(* CODESYS project Tc3_Physics.library
   TcLibraryId: Beckhoff Automation GmbH|Tc3_Physics|3.4.67.0
   Company: Beckhoff Automation GmbH
   DefaultNamespace: Tc3_Physics
   Version: 3.4.67.0
   Placeholder: Tc3_Physics
   Title: Tc3_Physics

Project tree, tasks and I/O mapping:
  Version/
    global variables Global_Version
  POUs/
    _Internal/
      function block IPlcGeometry2D [ST]: FB_init, FB_exit
      function block IPlcDynamicConstraint [ST]: FB_init, FB_exit
    Spatial/
      Positions/
        function block PositionXY [ST]: FB_init, FB_reinit, FB_exit, SetZero, SetValues, SetValuesXY, SetValuesRP, SetValuesXYReferenceId, GetRadius, GetPhi, Invert, ConcatenateWith, ShiftByXY, x, y, ReferenceId
        function block PositionXYC [ST]: FB_init, FB_reinit, FB_exit, SetZero, SetValues, SetValuesXY, SetValuesXYC, SetValuesXYCReferenceId, Invert, ConcatenateWith, StepByLocalXY, ShiftByXY, TurnByC, Transform, x, y, c, ReferenceId
    Dynamics/
      function block DynamicConstraint_Container [ST]: FB_init, FB_exit, Clear, AddConstraint, AddConstraintByReference, Count
      function block DynamicConstraint_CartesianXY [ST]: FB_init, FB_exit, SetValuesVAJ, V, A, J
      function block DynamicConstraint_CartesianXYZ [ST]: FB_init, FB_exit, SetValuesVAJ, V, A, J
      function block DynamicConstraint_PathXY [ST]: FB_init, FB_exit, SetValuesVADJ, V, A, D, J
      function block DynamicConstraint_PathXYZ [ST]: FB_init, FB_exit, SetValuesVADJ, V, A, D, J
      function block DynamicConstraint_Coordinates [ST]: FB_init, FB_exit, AddLimit, SetLimit, RemoveLimit, Clear, GetV, GetA, GetD, GetJ, Count
    Coordinates/
      function GetMcsCoordinateType [ST]
      function GetUninterpretedCoordinateType [ST]
      function GetAcsCoordinateType [ST]
  DUTs/
    Enumerations/
      data type E_RotationCoordinates
      data type E_CoordCategory
      data type E_McsCoordType
    data type CoordinateType
  GVLs/
    global variables GVL
*)

// DUTs/CoordinateType

(* Coordinate type. Use provided constants such as Coord_Mcs_X or factory functions such as GetMcsCoordinateType for creation. *)
	{attribute 'TcIecLibraryType'}
TYPE CoordinateType : 
	STRUCT
		(* Reserved. *)
		{attribute 'hide'}
		_reserved0 : ULINT := 0;
	END_STRUCT
END_TYPE

// DUTs/Enumerations/E_RotationCoordinates

(* 
    Enumeration of rotation conventions. 
    The order of letters defines the order of rotation around local axes.
    This also defines order in which user should program rotation values.
   *)
	{attribute 'TcIecLibraryType'}
{attribute 'qualified_only'}
{attribute 'strict'}
{attribute 'to_string'}
TYPE E_RotationCoordinates : (
	ABC:=0, 	(* ABC *)
	ACB:=1, 	(* ACB *)
	BCA:=2, 	(* BCA *)
	BAC:=3, 	(* BAC *)
	CAB:=4, 	(* CAB *)
	CBA:=5, 	(* CBA *)
	ABA:=6, 	(* ABA *)
	ACA:=7, 	(* ACA *)
	BCB:=8, 	(* BCB *)
	BAB:=9, 	(* BAB *)
	CAC:=10, 	(* CAC *)
	CBC:=11	(* CBC *)
) UDINT;
END_TYPE

// DUTs/Enumerations/E_CoordCategory

(* 
    Enumeration coordinate categories.
   *)
	{attribute 'TcIecLibraryType'}
{attribute 'qualified_only'}
{attribute 'strict'}
{attribute 'to_string'}
TYPE E_CoordCategory : (
	Invalid:=16#0, 	(* Invalid *)
	MCS:=16#1, 	(* MCS *)
	ACS:=16#2, 	(* ACS *)
	Uninterpreted:=16#3	(* Uninterpreted *)
) UDINT;
END_TYPE

// DUTs/Enumerations/E_McsCoordType

(* 
    Enumeration of MCS coordinate types.
   *)
	{attribute 'TcIecLibraryType'}
{attribute 'qualified_only'}
{attribute 'strict'}
{attribute 'to_string'}
TYPE E_McsCoordType : (
	Invalid:=16#0, 	(* Invalid *)
	X:=16#11, 	(* X *)
	Y:=16#21, 	(* Y *)
	Z:=16#31, 	(* Z *)
	A1:=16#41, 	(* A1 *)
	A2:=16#42, 	(* A2 *)
	A3:=16#43, 	(* A3 *)
	B1:=16#51, 	(* B1 *)
	B2:=16#52, 	(* B2 *)
	B3:=16#53, 	(* B3 *)
	C1:=16#61, 	(* C1 *)
	C2:=16#62, 	(* C2 *)
	C3:=16#63	(* C3 *)
) UDINT;
END_TYPE

// Version/Global_Version
{attribute 'TcGenerated'}
// This function has been automatically generated from the project information.
VAR_GLOBAL CONSTANT
	{attribute 'const_non_replaced'}
	{attribute 'linkalways'}
	stLibVersion_Tc3_Physics : ST_LibVersion := (iMajor := 3, iMinor := 4, iBuild := 67, iRevision := 0, sVersion := '3.4.67.0');
	{attribute 'const_non_replaced'}
	{attribute 'linkalways'}
	sLibraryId_Tc3_Physics : String := 'Beckhoff Automation GmbH|Tc3_Physics|3.4.67.0';
END_VAR

// GVLs/GVL

	{attribute 'external_name' := 'GVL_GUID_33C55D4C_0C6D_4080_813F_F3548CAD353B'}
VAR_GLOBAL CONSTANT
		Coord_Mcs_X	:	CoordinateType := GetMcsCoordinateType(E_McsCoordType.X);
		Coord_Mcs_Y	:	CoordinateType := GetMcsCoordinateType(E_McsCoordType.Y);
		Coord_Mcs_Z	:	CoordinateType := GetMcsCoordinateType(E_McsCoordType.Z);
		Coord_Mcs_A1	:	CoordinateType := GetMcsCoordinateType(E_McsCoordType.A1);
		Coord_Mcs_A2	:	CoordinateType := GetMcsCoordinateType(E_McsCoordType.A2);
		Coord_Mcs_A3	:	CoordinateType := GetMcsCoordinateType(E_McsCoordType.A3);
		Coord_Mcs_B1	:	CoordinateType := GetMcsCoordinateType(E_McsCoordType.B1);
		Coord_Mcs_B2	:	CoordinateType := GetMcsCoordinateType(E_McsCoordType.B2);
		Coord_Mcs_B3	:	CoordinateType := GetMcsCoordinateType(E_McsCoordType.B3);
		Coord_Mcs_C1	:	CoordinateType := GetMcsCoordinateType(E_McsCoordType.C1);
		Coord_Mcs_C2	:	CoordinateType := GetMcsCoordinateType(E_McsCoordType.C2);
		Coord_Mcs_C3	:	CoordinateType := GetMcsCoordinateType(E_McsCoordType.C3);
		Coord_Uninterpreted1	:	CoordinateType := GetUninterpretedCoordinateType(1);
		Coord_Uninterpreted2	:	CoordinateType := GetUninterpretedCoordinateType(2);
		Coord_Uninterpreted3	:	CoordinateType := GetUninterpretedCoordinateType(3);
		Coord_Uninterpreted4	:	CoordinateType := GetUninterpretedCoordinateType(4);
		Coord_Uninterpreted5	:	CoordinateType := GetUninterpretedCoordinateType(5);
		Coord_Uninterpreted6	:	CoordinateType := GetUninterpretedCoordinateType(6);
		Coord_Uninterpreted7	:	CoordinateType := GetUninterpretedCoordinateType(7);
		Coord_Uninterpreted8	:	CoordinateType := GetUninterpretedCoordinateType(8);
		Coord_Acs1	:	CoordinateType := GetAcsCoordinateType(1);
		Coord_Acs2	:	CoordinateType := GetAcsCoordinateType(2);
		Coord_Acs3	:	CoordinateType := GetAcsCoordinateType(3);
		Coord_Acs4	:	CoordinateType := GetAcsCoordinateType(4);
		Coord_Acs5	:	CoordinateType := GetAcsCoordinateType(5);
		Coord_Acs6	:	CoordinateType := GetAcsCoordinateType(6);
	END_VAR

// POUs/_Internal/IPlcGeometry2D

	{attribute 'c++_compatible'}
	{attribute 'external_name' := 'IPlcGeometry2D_GUID_432B7521_EF05_1C03_897A_3B970F77C0D6'}
	{attribute 'TcIecLibraryType'}
	{attribute 'no_explicit_call' :='do not call this POU directly'}
	{attribute 'no_assign_warning'}
	(* Internal representation of an object in the planar space. *)
	FUNCTION_BLOCK IPlcGeometry2D
	VAR
		(* x-coordinate of the instance. *)
		px : LREAL;
		(* y-coordinate of the instance. *)
		py : LREAL;
		(* c-rotation of the instance given in degrees [°]. *)
		pc : LREAL;
		 {attribute 'hide'}
		_reserved1 : ARRAY [1..24] OF USINT;
	END_VAR
	VAR_OUTPUT
		(* ErrorCode for last method execution *)
		nErrorId : UDINT;
		(* Error during last method execution *)
		bError : BOOL;
	END_VAR
	VAR
		 {attribute 'hide'}
		_reserved2 : ARRAY [1..35] OF USINT;
	END_VAR


	(* Internal method *)
	{attribute 'hide'}
	METHOD FB_init : BOOL
	VAR_INPUT
		(*  if TRUE, the retain variables are initialized (warm start / cold start) *)
		bInitRetains : BOOL;
		(*  if TRUE, the instance afterwards gets moved into the copy code (online change) *)
		bInCopyCode : BOOL;
	END_VAR
END_METHOD


	(* Internal method *)
	{attribute 'hide'}
	METHOD FB_exit : BOOL
	VAR_INPUT
		(*  if TRUE, the exit method is called for exiting an instance that is copied afterwards (online change). *)
		bInCopyCode : BOOL;
	END_VAR
END_METHOD

END_FUNCTION_BLOCK

// POUs/_Internal/IPlcDynamicConstraint

	{attribute 'c++_compatible'}
	{attribute 'external_name' := 'IPlcDynamicConstraint_GUID_6C0A73A2_C983_14C5_9BC7_15048F604248'}
	{attribute 'TcIecLibraryType'}
	{attribute 'no_explicit_call' := 'do not call this POU directly'}
	{attribute 'no_assign_warning'}
	(* Internal representation of dynamic constraints. *)
	FUNCTION_BLOCK IPlcDynamicConstraint
	VAR
		{attribute 'hide'}
		_reserved0 : ULINT;
		 {attribute 'hide'}
		_reserved1 : UINT_0_32;
		 {attribute 'hide'}
		_reserved2 : ARRAY [1..4] OF UINT_8_16;
		 {attribute 'hide'}
		_reserved3 : ARRAY [1..20] OF USINT;
	END_VAR


	(* Internal method *)
	{attribute 'hide'}
	METHOD FB_init : BOOL
	VAR_INPUT
		(*  if TRUE, the retain variables are initialized (warm start / cold start) *)
		bInitRetains : BOOL;
		(*  if TRUE, the instance afterwards gets moved into the copy code (online change) *)
		bInCopyCode : BOOL;
	END_VAR
END_METHOD


	(* Internal method *)
	{attribute 'hide'}
	METHOD FB_exit : BOOL
	VAR_INPUT
		(*  if TRUE, the exit method is called for exiting an instance that is copied afterwards (online change). *)
		bInCopyCode : BOOL;
	END_VAR
END_METHOD

END_FUNCTION_BLOCK

// POUs/Dynamics/DynamicConstraint_Container

	{attribute 'c++_compatible'}
	{attribute 'external_name' := 'DynamicConstraint_Container_GUID_0829228B_5233_1C1E_8F00_79BA3B649C7B'}
	{attribute 'TcIecLibraryType'}
	{attribute 'no_explicit_call' := 'do not call this POU directly'}
	{attribute 'no_assign_warning'}
	(* A container for dynamic constraints. *)
	FUNCTION_BLOCK DynamicConstraint_Container EXTENDS IPlcDynamicConstraint


	(* Internal method *)
	{attribute 'hide'}
	METHOD FB_init : BOOL
	VAR_INPUT
		(*  if TRUE, the retain variables are initialized (warm start / cold start) *)
		bInitRetains : BOOL;
		(*  if TRUE, the instance afterwards gets moved into the copy code (online change) *)
		bInCopyCode : BOOL;
	END_VAR
END_METHOD


	(* Internal method *)
	{attribute 'hide'}
	METHOD FB_exit : BOOL
	VAR_INPUT
		(*  if TRUE, the exit method is called for exiting an instance that is copied afterwards (online change). *)
		bInCopyCode : BOOL;
	END_VAR
END_METHOD


	(* Removes all dynamic constraints from the container. *)
	METHOD Clear
END_METHOD


	(* Adds a copy of a dynamic constraint to the container. If the dynamic constraint changes afterwards, the value in the container will not reflect that change. *)
	METHOD AddConstraint
	VAR_INPUT
		(* A reference to the constraint to be added. *)
 {attribute 'GUID' := '6C0A73A2-C983-14C5-9BC7-15048F604248'}
				Constraint : REFERENCE TO IPlcDynamicConstraint;
	END_VAR
END_METHOD


	(* Adds a reference to a dynamic constraint to the container. If the dynamic constraint changes afterwards, the value in the container will reflect that change. *)
	METHOD AddConstraintByReference
	VAR_INPUT
		(* A reference to the constraint to be added. *)
 {attribute 'GUID' := '6C0A73A2-C983-14C5-9BC7-15048F604248'}
				Constraint : REFERENCE TO IPlcDynamicConstraint;
	END_VAR
END_METHOD


{attribute 'monitoring' := 'call'}
	PROPERTY Count : UDINT
GET
END_GET
END_PROPERTY

END_FUNCTION_BLOCK

// POUs/Dynamics/DynamicConstraint_CartesianXY

	{attribute 'c++_compatible'}
	{attribute 'external_name' := 'DynamicConstraint_CartesianXY_GUID_45D77D0C_DF69_1CCA_AAA6_5FE79B258E7C'}
	{attribute 'TcIecLibraryType'}
	{attribute 'no_explicit_call' := 'do not call this POU directly'}
	(* Dynamic constraint for movement in the XY-plane, including non-tangential effects. *)
	FUNCTION_BLOCK DynamicConstraint_CartesianXY EXTENDS IPlcDynamicConstraint 
	VAR
		 {attribute 'hide'}
		_reserved1_1 : ARRAY [1..8] OF USINT;
	END_VAR


	(* Internal method *)
	{attribute 'hide'}
	METHOD FB_init : BOOL
	VAR_INPUT
		(*  if TRUE, the retain variables are initialized (warm start / cold start) *)
		bInitRetains : BOOL;
		(*  if TRUE, the instance afterwards gets moved into the copy code (online change) *)
		bInCopyCode : BOOL;
	END_VAR
END_METHOD


	(* Internal method *)
	{attribute 'hide'}
	METHOD FB_exit : BOOL
	VAR_INPUT
		(*  if TRUE, the exit method is called for exiting an instance that is copied afterwards (online change). *)
		bInCopyCode : BOOL;
	END_VAR
END_METHOD


	(* Set the dynamic limits of this instance. *)
	METHOD SetValuesVAJ
	VAR_INPUT
		(* Maximum velocity. *)
 {attribute 'GUID' := '0100FF8A-3F83-4535-990A-614CFBA4DA63'}
		 {attribute 'Namespace' := 'MC'}
				V : MC_LREAL;
		(* Maximum acceleration. *)
 {attribute 'GUID' := '0100FF8A-3F83-4535-990A-614CFBA4DA63'}
		 {attribute 'Namespace' := 'MC'}
				A : MC_LREAL;
		(* Maximum jerk. *)
 {attribute 'GUID' := '0100FF8A-3F83-4535-990A-614CFBA4DA63'}
		 {attribute 'Namespace' := 'MC'}
				J : MC_LREAL;
	END_VAR
END_METHOD


{attribute 'monitoring' := 'call'}
	PROPERTY V : MC_LREAL
GET
END_GET
SET
END_SET
END_PROPERTY


{attribute 'monitoring' := 'call'}
	PROPERTY A : MC_LREAL
GET
END_GET
SET
END_SET
END_PROPERTY


{attribute 'monitoring' := 'call'}
	PROPERTY J : MC_LREAL
GET
END_GET
SET
END_SET
END_PROPERTY

END_FUNCTION_BLOCK

// POUs/Dynamics/DynamicConstraint_CartesianXYZ

	{attribute 'c++_compatible'}
	{attribute 'external_name' := 'DynamicConstraint_CartesianXYZ_GUID_6A41E928_34B3_1C29_BA2B_E776EAC6142C'}
	{attribute 'TcIecLibraryType'}
	{attribute 'no_explicit_call' := 'do not call this POU directly'}
	(* Dynamic constraint for movement in the XYZ-space, including non-tangential effects. *)
	FUNCTION_BLOCK DynamicConstraint_CartesianXYZ EXTENDS IPlcDynamicConstraint 
	VAR
		 {attribute 'hide'}
		_reserved1_1 : ARRAY [1..8] OF USINT;
	END_VAR


	(* Internal method *)
	{attribute 'hide'}
	METHOD FB_init : BOOL
	VAR_INPUT
		(*  if TRUE, the retain variables are initialized (warm start / cold start) *)
		bInitRetains : BOOL;
		(*  if TRUE, the instance afterwards gets moved into the copy code (online change) *)
		bInCopyCode : BOOL;
	END_VAR
END_METHOD


	(* Internal method *)
	{attribute 'hide'}
	METHOD FB_exit : BOOL
	VAR_INPUT
		(*  if TRUE, the exit method is called for exiting an instance that is copied afterwards (online change). *)
		bInCopyCode : BOOL;
	END_VAR
END_METHOD


	(* Set the dynamic limits of this instance. *)
	METHOD SetValuesVAJ
	VAR_INPUT
		(* Maximum velocity. *)
 {attribute 'GUID' := '0100FF8A-3F83-4535-990A-614CFBA4DA63'}
		 {attribute 'Namespace' := 'MC'}
				V : MC_LREAL;
		(* Maximum acceleration. *)
 {attribute 'GUID' := '0100FF8A-3F83-4535-990A-614CFBA4DA63'}
		 {attribute 'Namespace' := 'MC'}
				A : MC_LREAL;
		(* Maximum jerk. *)
 {attribute 'GUID' := '0100FF8A-3F83-4535-990A-614CFBA4DA63'}
		 {attribute 'Namespace' := 'MC'}
				J : MC_LREAL;
	END_VAR
END_METHOD


{attribute 'monitoring' := 'call'}
	PROPERTY V : MC_LREAL
GET
END_GET
SET
END_SET
END_PROPERTY


{attribute 'monitoring' := 'call'}
	PROPERTY A : MC_LREAL
GET
END_GET
SET
END_SET
END_PROPERTY


{attribute 'monitoring' := 'call'}
	PROPERTY J : MC_LREAL
GET
END_GET
SET
END_SET
END_PROPERTY

END_FUNCTION_BLOCK

// POUs/Dynamics/DynamicConstraint_PathXY

	{attribute 'c++_compatible'}
	{attribute 'external_name' := 'DynamicConstraint_PathXY_GUID_C03A5F50_C097_1CA1_90CF_4DB7CF7C4E51'}
	{attribute 'TcIecLibraryType'}
	{attribute 'no_explicit_call' := 'do not call this POU directly'}
	{attribute 'no_assign_warning'}
	(* One dimensional dynamic constraint along the XY-components of a path, ignoring non-tangential effects. *)
	FUNCTION_BLOCK DynamicConstraint_PathXY EXTENDS IPlcDynamicConstraint 
	VAR
		 {attribute 'hide'}
		_reserved1_1 : ARRAY [1..8] OF USINT;
	END_VAR


	(* Internal method *)
	{attribute 'hide'}
	METHOD FB_init : BOOL
	VAR_INPUT
		(*  if TRUE, the retain variables are initialized (warm start / cold start) *)
		bInitRetains : BOOL;
		(*  if TRUE, the instance afterwards gets moved into the copy code (online change) *)
		bInCopyCode : BOOL;
	END_VAR
END_METHOD


	(* Internal method *)
	{attribute 'hide'}
	METHOD FB_exit : BOOL
	VAR_INPUT
		(*  if TRUE, the exit method is called for exiting an instance that is copied afterwards (online change). *)
		bInCopyCode : BOOL;
	END_VAR
END_METHOD


	(* Set the dynamic limits of this instance. *)
	METHOD SetValuesVADJ
	VAR_INPUT
		(* Maximum velocity. *)
 {attribute 'GUID' := '0100FF8A-3F83-4535-990A-614CFBA4DA63'}
		 {attribute 'Namespace' := 'MC'}
				V : MC_LREAL;
		(* Maximum acceleration. *)
 {attribute 'GUID' := '0100FF8A-3F83-4535-990A-614CFBA4DA63'}
		 {attribute 'Namespace' := 'MC'}
				A : MC_LREAL;
		(* Maximum deceleration. *)
 {attribute 'GUID' := '0100FF8A-3F83-4535-990A-614CFBA4DA63'}
		 {attribute 'Namespace' := 'MC'}
				D : MC_LREAL;
		(* Maximum jerk. *)
 {attribute 'GUID' := '0100FF8A-3F83-4535-990A-614CFBA4DA63'}
		 {attribute 'Namespace' := 'MC'}
				J : MC_LREAL;
	END_VAR
END_METHOD


{attribute 'monitoring' := 'call'}
	PROPERTY V : MC_LREAL
GET
END_GET
SET
END_SET
END_PROPERTY


{attribute 'monitoring' := 'call'}
	PROPERTY A : MC_LREAL
GET
END_GET
SET
END_SET
END_PROPERTY


{attribute 'monitoring' := 'call'}
	PROPERTY D : MC_LREAL
GET
END_GET
SET
END_SET
END_PROPERTY


{attribute 'monitoring' := 'call'}
	PROPERTY J : MC_LREAL
GET
END_GET
SET
END_SET
END_PROPERTY

END_FUNCTION_BLOCK

// POUs/Dynamics/DynamicConstraint_PathXYZ

	{attribute 'c++_compatible'}
	{attribute 'external_name' := 'DynamicConstraint_PathXYZ_GUID_95DC28DE_ABD8_106C_A9BB_995010C861A8'}
	{attribute 'TcIecLibraryType'}
	{attribute 'no_explicit_call' := 'do not call this POU directly'}
	(* One dimensional dynamic constraint along the XYZ-components of a path, ignoring non-tangential effects. *)
	FUNCTION_BLOCK DynamicConstraint_PathXYZ EXTENDS IPlcDynamicConstraint 
	VAR
		 {attribute 'hide'}
		_reserved1_1 : ARRAY [1..8] OF USINT;
	END_VAR


	(* Internal method *)
	{attribute 'hide'}
	METHOD FB_init : BOOL
	VAR_INPUT
		(*  if TRUE, the retain variables are initialized (warm start / cold start) *)
		bInitRetains : BOOL;
		(*  if TRUE, the instance afterwards gets moved into the copy code (online change) *)
		bInCopyCode : BOOL;
	END_VAR
END_METHOD


	(* Internal method *)
	{attribute 'hide'}
	METHOD FB_exit : BOOL
	VAR_INPUT
		(*  if TRUE, the exit method is called for exiting an instance that is copied afterwards (online change). *)
		bInCopyCode : BOOL;
	END_VAR
END_METHOD


	(* Set the dynamic limits of this instance. *)
	METHOD SetValuesVADJ
	VAR_INPUT
		(* Maximum velocity. *)
 {attribute 'GUID' := '0100FF8A-3F83-4535-990A-614CFBA4DA63'}
		 {attribute 'Namespace' := 'MC'}
				V : MC_LREAL;
		(* Maximum acceleration. *)
 {attribute 'GUID' := '0100FF8A-3F83-4535-990A-614CFBA4DA63'}
		 {attribute 'Namespace' := 'MC'}
				A : MC_LREAL;
		(* Maximum deceleration. *)
 {attribute 'GUID' := '0100FF8A-3F83-4535-990A-614CFBA4DA63'}
		 {attribute 'Namespace' := 'MC'}
				D : MC_LREAL;
		(* Maximum jerk. *)
 {attribute 'GUID' := '0100FF8A-3F83-4535-990A-614CFBA4DA63'}
		 {attribute 'Namespace' := 'MC'}
				J : MC_LREAL;
	END_VAR
END_METHOD


{attribute 'monitoring' := 'call'}
	PROPERTY V : MC_LREAL
GET
END_GET
SET
END_SET
END_PROPERTY


{attribute 'monitoring' := 'call'}
	PROPERTY A : MC_LREAL
GET
END_GET
SET
END_SET
END_PROPERTY


{attribute 'monitoring' := 'call'}
	PROPERTY D : MC_LREAL
GET
END_GET
SET
END_SET
END_PROPERTY


{attribute 'monitoring' := 'call'}
	PROPERTY J : MC_LREAL
GET
END_GET
SET
END_SET
END_PROPERTY

END_FUNCTION_BLOCK

// POUs/Dynamics/DynamicConstraint_Coordinates

	{attribute 'c++_compatible'}
	{attribute 'external_name' := 'DynamicConstraint_Coordinates_GUID_87FCCBE8_9B60_1095_89B3_AB2B0576CBCB'}
	{attribute 'TcIecLibraryType'}
	{attribute 'no_explicit_call' := 'do not call this POU directly'}
	{attribute 'no_assign_warning'}
	(* Dynamic constraints for individual coordinates. *)
	FUNCTION_BLOCK DynamicConstraint_Coordinates EXTENDS IPlcDynamicConstraint


	(* Internal method *)
	{attribute 'hide'}
	METHOD FB_init : BOOL
	VAR_INPUT
		(*  if TRUE, the retain variables are initialized (warm start / cold start) *)
		bInitRetains : BOOL;
		(*  if TRUE, the instance afterwards gets moved into the copy code (online change) *)
		bInCopyCode : BOOL;
	END_VAR
END_METHOD


	(* Internal method *)
	{attribute 'hide'}
	METHOD FB_exit : BOOL
	VAR_INPUT
		(*  if TRUE, the exit method is called for exiting an instance that is copied afterwards (online change). *)
		bInCopyCode : BOOL;
	END_VAR
END_METHOD


	(* Adds limits for a specific coordinate. If the coordinate is already limited, limits are merged. *)
	METHOD AddLimit
	VAR_INPUT
		(* Coordinate type. E.g. Coord_Mcs_X, Coord_Mcs_Y, ... *)
 {attribute 'GUID' := 'ABF37E9D-1614-4226-99CD-162368D15A32'}
				Coordinate : CoordinateType;
		(* Maximum velocity. *)
 {attribute 'GUID' := '0100FF8A-3F83-4535-990A-614CFBA4DA63'}
		 {attribute 'Namespace' := 'MC'}
				V : MC_LREAL;
		(* Maximum acceleration. *)
 {attribute 'GUID' := '0100FF8A-3F83-4535-990A-614CFBA4DA63'}
		 {attribute 'Namespace' := 'MC'}
				A : MC_LREAL;
		(* Maximum deceleration. *)
 {attribute 'GUID' := '0100FF8A-3F83-4535-990A-614CFBA4DA63'}
		 {attribute 'Namespace' := 'MC'}
				D : MC_LREAL;
		(* Maximum jerk. *)
 {attribute 'GUID' := '0100FF8A-3F83-4535-990A-614CFBA4DA63'}
		 {attribute 'Namespace' := 'MC'}
				J : MC_LREAL;
	END_VAR
END_METHOD


	(* Sets limits for a specific coordinate. If the coordinate is already limited, existing limits are overwritten. *)
	METHOD SetLimit
	VAR_INPUT
		(* Coordinate type. E.g. Coord_Mcs_X, Coord_Mcs_Y, ... *)
 {attribute 'GUID' := 'ABF37E9D-1614-4226-99CD-162368D15A32'}
				Coordinate : CoordinateType;
		(* Maximum velocity. *)
 {attribute 'GUID' := '0100FF8A-3F83-4535-990A-614CFBA4DA63'}
		 {attribute 'Namespace' := 'MC'}
				V : MC_LREAL;
		(* Maximum acceleration. *)
 {attribute 'GUID' := '0100FF8A-3F83-4535-990A-614CFBA4DA63'}
		 {attribute 'Namespace' := 'MC'}
				A : MC_LREAL;
		(* Maximum deceleration. *)
 {attribute 'GUID' := '0100FF8A-3F83-4535-990A-614CFBA4DA63'}
		 {attribute 'Namespace' := 'MC'}
				D : MC_LREAL;
		(* Maximum jerk. *)
 {attribute 'GUID' := '0100FF8A-3F83-4535-990A-614CFBA4DA63'}
		 {attribute 'Namespace' := 'MC'}
				J : MC_LREAL;
	END_VAR
END_METHOD


	(* Removes limits for a specific coordinate. *)
	METHOD RemoveLimit
	VAR_INPUT
		(* Coordinate type. E.g. Coord_Mcs_X, Coord_Mcs_Y, ... *)
 {attribute 'GUID' := 'ABF37E9D-1614-4226-99CD-162368D15A32'}
				Coordinate : CoordinateType;
	END_VAR
END_METHOD


	(* Removes limits for all coordinates. *)
	METHOD Clear
END_METHOD


	(* Gets the contained velocity limit for a specific coordinate. If no limits for the coordinate are set, returns MC_INVALID. *)
	METHOD GetV : MC_LREAL
	VAR_INPUT
		(* Coordinate type. E.g. Coord_Mcs_X, Coord_Mcs_Y, ... *)
 {attribute 'GUID' := 'ABF37E9D-1614-4226-99CD-162368D15A32'}
				Coordinate : CoordinateType;
	END_VAR
END_METHOD


	(* Gets the contained acceleration limit for a specific coordinate. If no limits for the coordinate are set, returns MC_INVALID. *)
	METHOD GetA : MC_LREAL
	VAR_INPUT
		(* Coordinate type. E.g. Coord_Mcs_X, Coord_Mcs_Y, ... *)
 {attribute 'GUID' := 'ABF37E9D-1614-4226-99CD-162368D15A32'}
				Coordinate : CoordinateType;
	END_VAR
END_METHOD


	(* Gets the contained deceleration limit for a specific coordinate. If no limits for the coordinate are set, returns MC_INVALID. *)
	METHOD GetD : MC_LREAL
	VAR_INPUT
		(* Coordinate type. E.g. Coord_Mcs_X, Coord_Mcs_Y, ... *)
 {attribute 'GUID' := 'ABF37E9D-1614-4226-99CD-162368D15A32'}
				Coordinate : CoordinateType;
	END_VAR
END_METHOD


	(* Gets the contained jerk limit for a specific coordinate. If no limits for the coordinate are set, returns MC_INVALID. *)
	METHOD GetJ : MC_LREAL
	VAR_INPUT
		(* Coordinate type. E.g. Coord_Mcs_X, Coord_Mcs_Y, ... *)
 {attribute 'GUID' := 'ABF37E9D-1614-4226-99CD-162368D15A32'}
				Coordinate : CoordinateType;
	END_VAR
END_METHOD


{attribute 'monitoring' := 'call'}
	PROPERTY Count : UDINT
GET
END_GET
END_PROPERTY

END_FUNCTION_BLOCK

// POUs/Coordinates/GetMcsCoordinateType

	{attribute 'TcIecLibraryType'}
	{attribute 'external_name' := 'GetMcsCoordinateType_GUID_369DBA31_787B_1B81_8BF3_86CFF64C1E07'}
	(* Creates a CoordinateType FB from E_McsCoordType. *)
	FUNCTION GetMcsCoordinateType : CoordinateType
	VAR_INPUT
		mcsType	:	E_McsCoordType;	(* Mcs coordinate type. *)
	END_VAR

END_FUNCTION

// POUs/Coordinates/GetUninterpretedCoordinateType

	{attribute 'TcIecLibraryType'}
	{attribute 'external_name' := 'GetUninterpretedCoordinateType_GUID_3E2E03A5_07C2_19F8_A0C2_0F94EA0A56A4'}
	(* Creates a CoordinateType FB from an index. *)
	FUNCTION GetUninterpretedCoordinateType : CoordinateType
	VAR_INPUT
		index	:	UDINT;	(* Uninterpreted coordinate type. *)
	END_VAR

END_FUNCTION

// POUs/Coordinates/GetAcsCoordinateType

	{attribute 'TcIecLibraryType'}
	{attribute 'external_name' := 'GetAcsCoordinateType_GUID_7DE58953_274B_1D87_B664_E9E87F11C35C'}
	(* Creates a CoordinateType FB from an index. *)
	FUNCTION GetAcsCoordinateType : CoordinateType
	VAR_INPUT
		index	:	UDINT;	(* Acs coordinate type. *)
	END_VAR

END_FUNCTION

// POUs/Spatial/Positions/PositionXY

	{attribute 'c++_compatible'}
	{attribute 'external_name' := 'PositionXY_GUID_97A8C469_9E33_1367_BD2B_4B487B94CC01'}
	{attribute 'TcIecLibraryType'}
	{attribute 'no_explicit_call' :='do not call this POU directly'}
	{attribute 'no_assign_warning'}
	(* Position in the 2D Cartesian space. *)
	FUNCTION_BLOCK PositionXY EXTENDS IPlcGeometry2D


	(* Internal method *)
	{attribute 'hide'}
	METHOD FB_init : BOOL
	VAR_INPUT
		(*  if TRUE, the retain variables are initialized (warm start / cold start) *)
		bInitRetains : BOOL;
		(*  if TRUE, the instance afterwards gets moved into the copy code (online change) *)
		bInCopyCode : BOOL;
	END_VAR
END_METHOD


	(* Internal method *)
	{attribute 'hide'}
	METHOD FB_reinit : BOOL
END_METHOD


	(* Internal method *)
	{attribute 'hide'}
	METHOD FB_exit : BOOL
	VAR_INPUT
		(*  if TRUE, the exit method is called for exiting an instance that is copied afterwards (online change). *)
		bInCopyCode : BOOL;
	END_VAR
END_METHOD


	(* Set the coordinates of this position to '0.0'. *)
	METHOD SetZero
END_METHOD


	(* Set the coordinates of this position. *)
	METHOD SetValues
	VAR_IN_OUT
		(* The coordinate values to set. *)
 {attribute 'GUID' := '97A8C469-9E33-1367-BD2B-4B487B94CC01'}
				positionXY : PositionXY;
	END_VAR
END_METHOD


	(* Set the xy-coordinates of this position. *)
	METHOD SetValuesXY
	VAR_INPUT
		(* x-component of the position. *)
		x : LREAL;
		(* y-component of the position. *)
		y : LREAL;
	END_VAR
END_METHOD


	(* Set the components of this position in polar coordinates. *)
	METHOD SetValuesRP
	VAR_INPUT
		(* Distance from the origin. *)
		radius : LREAL;
		(* Polar angle of this position in degrees [°]. *)
		phi : LREAL;
	END_VAR
END_METHOD


	(* Set the xy-coordinates of this position and the reference id. *)
	METHOD SetValuesXYReferenceId
	VAR_INPUT
		(* x-component of the position. *)
		x : LREAL;
		(* y-component of the position. *)
		y : LREAL;
		(* reference id of the position. *)
 {attribute 'GUID' := '18071995-0000-0000-0000-00000000000F'}
				ReferenceId : OTCID;
	END_VAR
END_METHOD


	(* Get the distance from the origin. *)
	METHOD GetRadius : LREAL
END_METHOD


	(* Get the polar angle scaled in degrees [°]. *)
	METHOD GetPhi : LREAL
END_METHOD


	(* Invert this position. *)
	METHOD Invert
END_METHOD


	(* Concatenate with a 2nd position. *)
	METHOD ConcatenateWith
	VAR_IN_OUT
		(* The 2nd position to concatenate with. *)
 {attribute 'GUID' := '97A8C469-9E33-1367-BD2B-4B487B94CC01'}
				position : PositionXY;
	END_VAR
END_METHOD


	(* Displace the components of this position. *)
	METHOD ShiftByXY
	VAR_INPUT
		(* Shift of the x-component of this position. *)
		dx : LREAL;
		(* Shift of the y-component of this position. *)
		dy : LREAL;
	END_VAR
END_METHOD


	PROPERTY x : LREAL
GET
END_GET
SET
END_SET
END_PROPERTY


	PROPERTY y : LREAL
GET
END_GET
SET
END_SET
END_PROPERTY


{attribute 'monitoring' := 'call'}
	PROPERTY ReferenceId : OTCID
GET
END_GET
SET
END_SET
END_PROPERTY

END_FUNCTION_BLOCK

// POUs/Spatial/Positions/PositionXYC

	{attribute 'c++_compatible'}
	{attribute 'external_name' := 'PositionXYC_GUID_12927DD4_F3D1_1B21_A804_08BCF50529B3'}
	{attribute 'TcIecLibraryType'}
	{attribute 'no_explicit_call' :='do not call this POU directly'}
	{attribute 'no_assign_warning'}
	(* A position in the xy-plane with an in-plane direction c. *)
	FUNCTION_BLOCK PositionXYC EXTENDS IPlcGeometry2D


	(* Internal method *)
	{attribute 'hide'}
	METHOD FB_init : BOOL
	VAR_INPUT
		(*  if TRUE, the retain variables are initialized (warm start / cold start) *)
		bInitRetains : BOOL;
		(*  if TRUE, the instance afterwards gets moved into the copy code (online change) *)
		bInCopyCode : BOOL;
	END_VAR
END_METHOD


	(* Internal method *)
	{attribute 'hide'}
	METHOD FB_reinit : BOOL
END_METHOD


	(* Internal method *)
	{attribute 'hide'}
	METHOD FB_exit : BOOL
	VAR_INPUT
		(*  if TRUE, the exit method is called for exiting an instance that is copied afterwards (online change). *)
		bInCopyCode : BOOL;
	END_VAR
END_METHOD


	(* Set the components of this vector to '0.0'. *)
	METHOD SetZero
END_METHOD


	(* Set the components of this position. *)
	METHOD SetValues
	VAR_IN_OUT
		(* The values to set. *)
 {attribute 'GUID' := '12927DD4-F3D1-1B21-A804-08BCF50529B3'}
				positionXYC : PositionXYC;
	END_VAR
END_METHOD


	(* Set the spatial components of this position. *)
	METHOD SetValuesXY
	VAR_INPUT
		(* x-component of the position. *)
		x : LREAL;
		(* y-component of the position. *)
		y : LREAL;
	END_VAR
END_METHOD


	(* Set the components of this position. *)
	METHOD SetValuesXYC
	VAR_INPUT
		(* x-component of the position. *)
		x : LREAL;
		(* y-component of the position. *)
		y : LREAL;
		(* c-component of the position scaled in degrees [°]. *)
		c : LREAL;
	END_VAR
END_METHOD


	(* Set the components of this position. *)
	METHOD SetValuesXYCReferenceId
	VAR_INPUT
		(* x-component of the position. *)
		x : LREAL;
		(* y-component of the position. *)
		y : LREAL;
		(* c-component of the position scaled in degrees [°]. *)
		c : LREAL;
		(* reference id of the position. *)
 {attribute 'GUID' := '18071995-0000-0000-0000-00000000000F'}
				ReferenceId : OTCID;
	END_VAR
END_METHOD


	(* Invert this position. *)
	METHOD Invert
END_METHOD


	(* Multiply this position by a 2nd from the right. *)
	METHOD ConcatenateWith
	VAR_IN_OUT
		(* The position to concatenate with. *)
 {attribute 'GUID' := '12927DD4-F3D1-1B21-A804-08BCF50529B3'}
				position : PositionXYC;
	END_VAR
END_METHOD


	(* Apply a local step in respect to the local coordinate frame without changing the orientation. *)
	METHOD StepByLocalXY
	VAR_INPUT
		(* The displacement within the local x-direction. *)
		dx : LREAL;
		(* The displacement within the local y-direction. *)
		dy : LREAL;
	END_VAR
END_METHOD


	(* Displace the components of this position. *)
	METHOD ShiftByXY
	VAR_INPUT
		(* Shift of the x-component of this position. *)
		dx : LREAL;
		(* Shift of the y-component of this position. *)
		dy : LREAL;
	END_VAR
END_METHOD


	(* Rotate the attached orientation without changing the Cartesian coordinates. *)
	METHOD TurnByC
	VAR_INPUT
		(* Angular displacement given in degrees [°]. *)
		dc : LREAL;
	END_VAR
END_METHOD


	(* Place a PositionXY into the coordinate system referenced by this position. *)
	METHOD Transform
	VAR_IN_OUT
		(* Position to transform. *)
 {attribute 'GUID' := '97A8C469-9E33-1367-BD2B-4B487B94CC01'}
				positionXY : PositionXY;
	END_VAR
END_METHOD


	PROPERTY x : LREAL
GET
END_GET
SET
END_SET
END_PROPERTY


	PROPERTY y : LREAL
GET
END_GET
SET
END_SET
END_PROPERTY


	PROPERTY c : LREAL
GET
END_GET
SET
END_SET
END_PROPERTY


{attribute 'monitoring' := 'call'}
	PROPERTY ReferenceId : OTCID
GET
END_GET
SET
END_SET
END_PROPERTY

END_FUNCTION_BLOCK
